ABB RobotStudio station: Tp2.rsstn

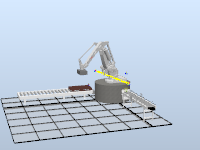
Station Tp2 (saved by RobotStudio 20.2.9116.0)
Controller Controlador1
  mechanical unit ROB_1: IRB660_180_315__01_2, 6 joints, base frame (0, 0, 1000) mm
Layout (positions relative to the parent item):
  - transporteCajas [part, from Equipment\Conveyor Guide 400.rslib] at (0, 1500, 0) mm, rotated rx 0 ry 0 rz 90 deg
  - Euro Pallet [graphiccomponentgroup, from Equipment\Euro Pallet.rslib] at (1000, -1425, 435) mm
    - Body 1 [part, from Equipment\Euro Pallet.rslib]
  - transportePallets [part, from Equipment\Conveyor 950 4000 h2.rslib] at (1000, -1500, 0) mm
  - IRB660_180_315__01_2 [mechanism, from Robots\IRB660_180_315__01.rslib] at (0, 0, 1000) mm; joint values [0.4196, 0.4368, 0.607, 0.4196] (rad or m)
  - ventosa_tool [mechanism] at (2018.58, 900.45, 1942.78) mm, rotated rx 180 ry 0 rz 180 deg
      TCP ventosa_tool at (0, 0, 200) mm
      links: ventosa
  - pedestal [part]
  - fuenteBloques [smart component] at (-200, 1500, 770) mm
      signals: DI agarrar, DO cajaLista, DI soltar
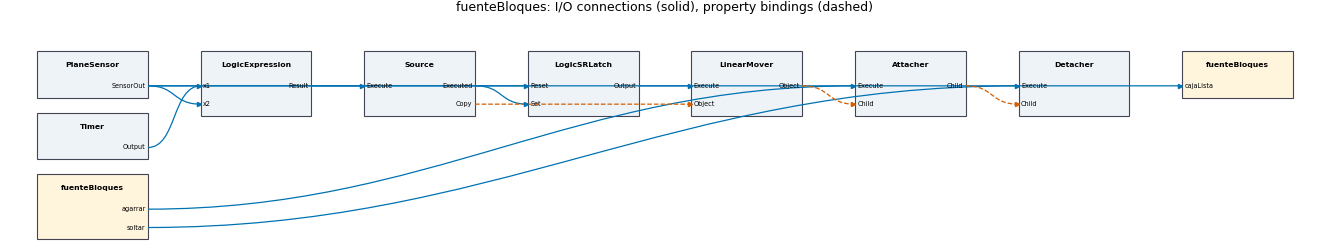
      connections:
        LogicSRLatch.Output -> LinearMover.Execute
        PlaneSensor.SensorOut -> LogicSRLatch.Reset
        Timer.Output -> LogicExpression.x1
        PlaneSensor.SensorOut -> LogicExpression.x2
        LogicExpression.Result -> Source.Execute
        Source.Executed -> LogicSRLatch.Set
        PlaneSensor.SensorOut -> fuenteBloques.cajaLista
        fuenteBloques.agarrar -> Attacher.Execute
        fuenteBloques.soltar -> Detacher.Execute
        LinearMover.Object => Attacher.Child
        Attacher.Child => Detacher.Child
        Source.Copy => LinearMover.Object
    - Source [smart component, from Components\Source.rslib]
        properties: Source=caja; Copy=(none); Parent=(none); Position=[0 2.5 0]; Orientation=[0 0 0]; Transient=true; PhysicsBehavior=0
    - Timer [smart component, from Components\Timer.rslib]
        properties: StartTime=0; Interval=5; Repeat=true; CurrentTime=11.4
    - LinearMover [smart component, from Components\LinearMover.rslib]
        properties: Object=(none); Direction=[0 2.5 0]; Speed=-0.8; Reference=Local; ReferenceObject=fuenteBloques
    - PlaneSensor [smart component, from Components\PlaneSensor.rslib]
        properties: Origin=[-0.1 0.00100000000000011 0]; Axis1=[0 0 0.2]; Axis2=[0.2 0 0]; SensedPart=(none)
      - _sensorPart_ [part]
    - Queue [smart component, from Components\Queue.rslib]
        properties: Back=(none); Front=(none); Queue=; NumberOfObjects=0
    - caja [part]
    - LogicSRLatch [smart component, from Components\LogicSRLatch.rslib]
    - LogicExpression [smart component, from Components\LogicExpression.rslib]
        properties: Expression=x1 AND NOT x2
    - Attacher [smart component, from Components\Attacher.rslib]
        properties: Parent=Detacher; Flange=0; Child=(none); Mount=false; Offset=[0 0 0]; Orientation=[0 0 0]
    - Detacher [smart component, from Components\Detacher.rslib]
        properties: Child=(none); KeepPosition=true
    - StopSimulation [smart component, from Components\StopSimulation.rslib]
    - StopSimulation_2 [smart component, from Components\StopSimulation.rslib]
Attachment: Euro Pallet is attached to transportePallets
Attachment: ventosa_tool is attached to IRB660_180_315__01_2 / Link6
Attachment: pistaCajas is attached to transporteCajas
Attachment: pistaPallets is attached to transportePallets
Station logic (signal -> signal, property => property):
  Controlador1.do_pick -> fuenteBloques.agarrar
  fuenteBloques.cajaLista -> Controlador1.cajaLista
  Controlador1.do_place -> fuenteBloques.soltar
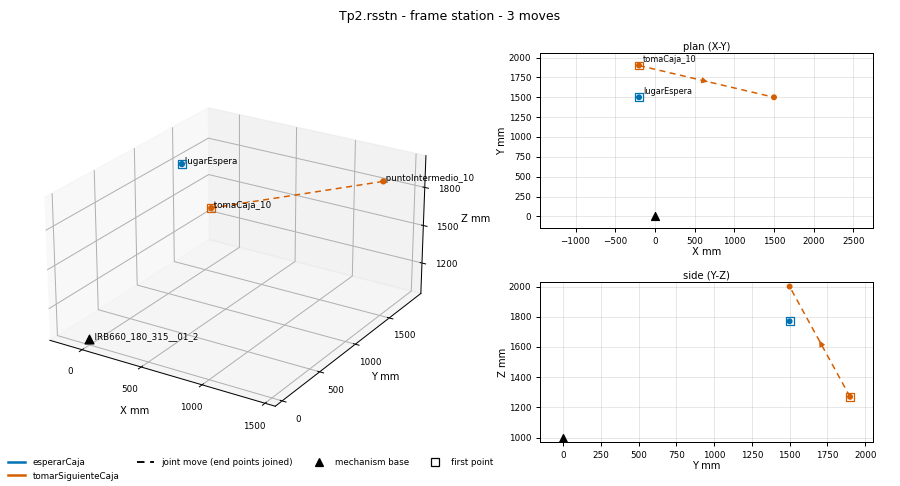
[picture p0: tool path of Tp2.rsstn in frame station, 3 of 3 moves have a stored position in this frame; points joined in program order, loops and branches not executed]
Targets, tools, work objects and paths stored in the station, written as RAPID:
! task T_ROB1
MODULE Module1
  PERS tooldata ventosa_tool:=[TRUE,[[0,0,200],[1,0,0,0]],[1,[0,0,1],[1,0,0,0],0,0,0]];
  PERS wobjdata pistaCajas:=[FALSE,TRUE,"",[[-200,1500,770],[0,0,1,0]],[[0,0,0],[1,0,0,0]]];
  PERS wobjdata pistaPallets:=[FALSE,TRUE,"",[[1000,-1425,579],[0,0,1,0]],[[0,0,0],[1,0,0,0]]];
  CONST robtarget lugarEspera:=[[0,0,-1000],[1,0,0,0],[0,0,0,0],[9E+09,9E+09,9E+09,9E+09,9E+09,9E+09]];
  CONST robtarget tomaCaja_10:=[[0,400,-500],[1,0,0,0],[0,0,0,0],[9E+09,9E+09,9E+09,9E+09,9E+09,9E+09]];
  CONST robtarget superficiePallet_10:=[[0,0,0],[1,0,0,0],[0,0,0,0],[9E+09,9E+09,9E+09,9E+09,9E+09,9E+09]];
  CONST robtarget puntoIntermedio_10:=[[1500,1500,2000],[0,0,1,0],[0,0,0,0],[9E+09,9E+09,9E+09,9E+09,9E+09,9E+09]];
  PROC main()
    SetDO do_pick,0;
    esperarCaja;
    tomarSiguienteCaja;
    esperarCaja;
  ENDPROC
  PROC esperarCaja()
    MoveJ lugarEspera,v1000,fine,ventosa_tool\WObj:=pistaCajas;
    WaitDI cajaLista,1;
  ENDPROC
  PROC tomarSiguienteCaja()
    MoveJ tomaCaja_10,v1000,fine,ventosa_tool\WObj:=pistaCajas;
    SetDO do_place,0;
    SetDO do_pick,1;
    MoveJ puntoIntermedio_10,v1000,z100,ventosa_tool\WObj:=wobj0;
  ENDPROC
ENDMODULE

